{attribute 'GeneratedUsingTerminal: EL3314-0030-0021'}
{attribute addProperty BoxType "EL3314-0030-0021"}
{attribute addProperty Id "EtcSlaveTerminalBaseTC_Inputs_Channel_1AT %I*TC_Inputs_Channel_204FE7509TC_Inputs_Channel_2AT %I*TC_Inputs_Channel_204FE7509TC_Inputs_Channel_3AT %I*TC_Inputs_Channel_204FE7509TC_Inputs_Channel_4AT %I*TC_Inputs_Channel_204FE7509WcStateAT %I*WcState_9091E0EB2InfoDataAT %I*InfoData_32EB74EA10"}
{attribute addProperty CRC "350323065"}
{attribute addProperty Size "48"}
TYPE EL3314_14E18179 EXTENDS EtcSlaveTerminalBase :
STRUCT
	{attribute addProperty Name "TC_Inputs_Channel_1"}
	TC_Inputs_Channel_1 : TC_Inputs_Channel_204FE750;
	{attribute addProperty Name "TC_Inputs_Channel_2"}
	TC_Inputs_Channel_2 : TC_Inputs_Channel_204FE750;
	{attribute addProperty Name "TC_Inputs_Channel_3"}
	TC_Inputs_Channel_3 : TC_Inputs_Channel_204FE750;
	{attribute addProperty Name "TC_Inputs_Channel_4"}
	TC_Inputs_Channel_4 : TC_Inputs_Channel_204FE750;
	{attribute addProperty Name "WcState"}
	WcState : WcState_9091E0EB;
	{attribute addProperty Name "InfoData"}
	InfoData : InfoData_32EB74EA;
END_STRUCT
END_TYPE

(* stored: Version 1.2.0.0, ProductVersion 3.1.4024.9
   DUT EL3314_14E18179: Id {0490fa9a-6484-4668-bd24-1086e4a47e03} *)
